// TIA Portal V17 export
// export: Created 2024-09-03T21:54:52.161181Z, ExportSetting WithDefaults, DisplayName Totally Integrated Automation Portal, DisplayVersion V17 Update 7, DisplayName TIA Portal Openness, DisplayVersion V17 Update 7, DisplayName TIA Portal Version Control Interface, DisplayVersion V17, DisplayName SINAMICS Startdrive Advanced, DisplayVersion V17 SP2, DisplayName SINAMICS Startdrive G110M, G120, G120C, G120D, G120P, G115D, DisplayVersion V17 SP2, DisplayName SINAMICS Startdrive G130, G150, S120, S150, SINAMICS MV, S210, DisplayVersion V17 SP2, DisplayName STEP 7 Professional, DisplayVersion V17 Update 7, DisplayName STEP 7 Safety, DisplayVersion V17 Update 6, DisplayName WinCC Advanced / Unified PC, DisplayVersion V17 Update 7
DATA_BLOCK "READER_MODEL"   // DB74
{ S7_Optimized_Access := 'TRUE' }
VERSION : 0.1
// stored: AutoNumber true, DBAccessibleFromOPCUA true, DBAccessibleFromWebserver true, IsOnlyStoredInLoadMemory false, IsRetainMemResEnabled false, IsWriteProtectedInAS false, MemoryReserve 100
   VAR RETAIN
      PRODUCT { S7_SetPoint := 'True'} : Array[0.."NumberOfProductionPrograms"] of "READER_PRODUCT";
   END_VAR
BEGIN
   PRODUCT[1..4].SIDE_RH.POSITION := 13;
   PRODUCT[1..4].SIDE_RH.LEN := 3;
   PRODUCT[1].SIDE_RH.STRING_LABEL := '336';
   PRODUCT[2].SIDE_RH.STRING_LABEL := '532';
   PRODUCT[3].SIDE_RH.STRING_LABEL := '336';
   PRODUCT[4].SIDE_RH.STRING_LABEL := '532';
   PRODUCT[1..4].SIDE_RH.READER_BYPASS := FALSE;
   PRODUCT[1..4].SIDE_LH.POSITION := 13;
   PRODUCT[1..4].SIDE_LH.LEN := 3;
   PRODUCT[1].SIDE_LH.STRING_LABEL := '328';
   PRODUCT[2].SIDE_LH.STRING_LABEL := '526';
   PRODUCT[3].SIDE_LH.STRING_LABEL := '328';
   PRODUCT[4].SIDE_LH.STRING_LABEL := '526';
   PRODUCT[1..4].SIDE_LH.READER_BYPASS := FALSE;
   PRODUCT[1..4].REAR_TUBE.POSITION := 13;
   PRODUCT[1..4].REAR_TUBE.LEN := 3;
   PRODUCT[1].REAR_TUBE.STRING_LABEL := '343';
   PRODUCT[2].REAR_TUBE.STRING_LABEL := '514';
   PRODUCT[3].REAR_TUBE.STRING_LABEL := '343';
   PRODUCT[4].REAR_TUBE.STRING_LABEL := '514';
   PRODUCT[1..4].REAR_TUBE.READER_BYPASS := FALSE;
   PRODUCT[1..2].FRONT_TUBE.POSITION := 13;
   PRODUCT[1..2].FRONT_TUBE.LEN := 3;
   PRODUCT[1..2].FRONT_TUBE.STRING_LABEL := '907';
   PRODUCT[1].FRONT_TUBE.READER_BYPASS := FALSE;
   PRODUCT[2..4].FRONT_TUBE.READER_BYPASS := TRUE;
   PRODUCT[1..2].NUM_TUBE := TRUE;
   PRODUCT[3].NUM_TUBE := FALSE;
END_DATA_BLOCK
